// Mitsubishi GX Works2 project: dataEx01   PLC: Q02/Q02H

PROGRAM MAIN
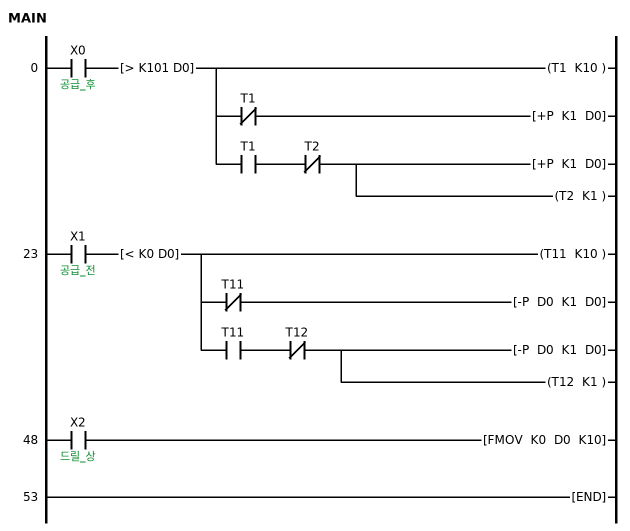
0     LD      X0  ; 공급_후
      AND>    K101 D0
      OUT     T1 K10
      MPS
      ANI     T1
      +P      K1 D0
      MPP
      AND     T1
      ANI     T2
      +P      K1 D0
      OUT     T2 K1
23    LD      X1  ; 공급_전
      AND<    K0 D0
      OUT     T11 K10
      MPS
      ANI     T11
      -P      D0 K1 D0
      MPP
      AND     T11
      ANI     T12
      -P      D0 K1 D0
      OUT     T12 K1
48    LD      X2  ; 드릴_상
      FMOV    K0 D0 K10
53    END
END_PROGRAM

// device comments not shown above
X3  ; 드릴_하
X4  ; 송출_후
X5  ; 송출_전
X6  ; 배출_후
X7  ; 배출_전
X8  ; 매거진
X9  ; 비금속
X0A  ; 금속
X10  ; PB1
X11  ; PB2
X12  ; PB3
Y20  ; 공급_전
Y21  ; 공급_후
Y22  ; 드릴_하강
Y23  ; 송출_전
Y24  ; 송출_후
Y25  ; 배출_전
Y26  ; 배출_후
Y27  ; 컨베어
Y28  ; 가공드
Y29  ; 적색
Y2A  ; 황색
Y2B  ; 녹색
